{attribute 'GeneratedUsingTerminal: EL6900-0000-0016'}
{attribute addProperty BoxType "EL6900-0000-0016"}
{attribute addProperty Id "ControlAT %Q*UINT2"}
{attribute addProperty CRC "3674028256"}
{attribute addProperty Size "2"}
TYPE DEVICE_Outputs_DAFD38E0 :
STRUCT
	{attribute addProperty Name "Control"}
	Control AT %Q* : UINT;
END_STRUCT
END_TYPE

(* stored: Version 1.2.0.0, ProductVersion 3.1.4024.9
   DUT DEVICE_Outputs_DAFD38E0: Id {bc58f254-7471-4ba1-aa59-dc27963a1032} *)
